// TIA Portal V19 export
DATA_BLOCK "DB_Fahr-Hubzeit"   // DB5
{ S7_Optimized_Access := 'FALSE' }
// stored: AutoNumber false
   VAR RETAIN
      FZ_Typ_Pos : Real := 1.0;   // Fahrzeit typisch Position zu Position
      FZ_Typ_Halt : Real := 5.0;   // Fahrzeit typisch für Positionierung
      UZ_typ : Real := 40.0;   // typische Umsetzzeit (für Zwischenschieben)
      HZ_Gestell_langsam : Real := 20.0;   // Hubzeit typisch für Gestelle bei langsamen Hub
      HZ_Gestell_schnell : Real := 15.0;   // Hubzeit typisch für Gestelle bei schnellen Hub
      HZ_Trommel_langsam : Real := 20.0;   // Hubzeit typisch für Trommeln bei langsamen Hub
      HZ_Trommel_schnell : Real := 15.0;   // Hubzeit typisch für Trommeln bei schnellen Hub
      SZ_Gestell_langsam : Real := 20.0;   // Senkzeit typisch für Gestelle bei langsamen Hub
      SZ_Gestell_schnell : Real := 15.0;   // Senkzeit typisch für Gestelle bei schnellen Hub
      SZ_Trommel_langsam : Real := 20.0;   // Senkzeit typisch für Trommeln bei langsamen Hub
      SZ_Trommel_schnell : Real := 15.0;   // Senkzeit typisch für Trommeln bei schnellen Hub
      TS_Zeit : Real := 0.0;   // Schwenkzeit Tropfwanne typisch
   END_VAR
BEGIN
END_DATA_BLOCK
